Fanuc KAREL source: kc00052.KL

-- PROVISIONAL review KL for V1013-1; original PC SHA256 59a8608078e209181223c6af16679c1e7fcb64aa9bab4861e9d6acceead57624
-- Incomplete behavior may be omitted. Consult companion uncertainty JSON. Do not deploy.
PROGRAM KC00052
%NOLOCKGROUP
BEGIN
  -- UNRESOLVED_PC offsets 5-39; opcodes 27,22,22,22,22,22,31
  -- UNRESOLVED_PC offsets 44-48; opcodes 7F
END KC00052
